TYPE "SinamicsCU_Warnings"
VERSION : 0.1
// Block: SinamicsCU_Warnings
   STRUCT
      CUWarning : Bool;
      CUSafetyMessagePresence : Bool;
   END_STRUCT;

END_TYPE
